TYPE BreakStopConfig :
STRUCT
	MaxTimeLeavingStop: TIME;
	DebounceTimePuckPresentOn: TIME;
	DebounceTimePuckPresentOff: TIME;
	DebounceTimeBufferFullOn: TIME;
	DebounceTimeBufferFullOff: TIME;
	TimeSpacingMinimum: TIME;
	EnableBufferArrivalFault: BOOL;
	BufferArrivalFaultTime: TIME;
END_STRUCT
END_TYPE

(* stored: Version 1.1.0.1, ProductVersion 3.1.4024.6
   DUT BreakStopConfig: Id {282fbd3e-6610-4a3e-8ffb-54d570dbc54a} *)
